// TIA Portal V21 export
VAR_GLOBAL   // PLC tag table "K_RicettaSpiedinatrice"
END_VAR
VAR_GLOBAL CONSTANT   // user constants
   K_DatoRicettaReal_Spiedinatrice_QuotaPrimoInserimentoStecchi : Int := 1;
   K_DatoRicettaReal_Spiedinatrice_NumeroFilePerLato : Int := 2;
   K_DatoRicettaReal_Spiedinatrice_DistanzaTraGliStecchi : Int := 3;
   K_DatoRicettaReal_Spiedinatrice_QuoteFileStecchiNelCubo : Int := 4;
   K_DatoRicettaReal_Spiedinatrice_AltezzaTotCubo : Int := 5;
END_VAR
